# EPICS alarm handler configuration: alh_files/mgnt_li23.alhConfig
GROUP NULL MGNT:LI23:1
   $COMMAND edm -x -eolc -noedit mgnt_li23_main.edl

$ALIAS LI23
$GUIDANCE
LI23 Magnets
   Group Name: MGNT:LI23:1
   Summary PV:  MGNT:LI23:1:STATSUMY
$END

   INCLUDE MGNT:LI23:1 ./mgnt_li23_lgps.alhConfig
   INCLUDE MGNT:LI23:1 ./mgnt_li23_quad.alhConfig
   INCLUDE MGNT:LI23:1 ./mgnt_li23_xcor.alhConfig
   INCLUDE MGNT:LI23:1 ./mgnt_li23_ycor.alhConfig
